// TIA Portal V20 export
FUNCTION_BLOCK "FB_PowerMeterSeq"   // FB92, SCL
{ S7_Optimized_Access := 'TRUE' }
// stored: AutoNumber false, MemoryReserve 100, SetENOAutomatically false
   VAR_INPUT
      iStartSeqCond : Bool;   // Start Sequence Conditions
      iJobReq : Bool;   // Job Request - From Main
      iPowerMeterHomePos : Bool;
      iPowerMeterWorkPos : Bool;
      iNC_Stopped : Bool;
      iPLC_DateAndTime : DTL;
      iStepPause : Bool;
      rMinValue : Real;
      rMaxValue : Real;
      iStopOption : Bool;
      rMeasureValue : Real;
      iMeasureDone : Bool;
   END_VAR
   VAR_OUTPUT
      oPowerMetertoHomeReq { ExternalAccessible := 'False'; ExternalVisible := 'False'; ExternalWritable := 'False'} : Bool;   // Shuttle Start Order - To FB_LoaderAxis
      oPowerMetertoWorkReq { ExternalAccessible := 'False'; ExternalVisible := 'False'; ExternalWritable := 'False'} : Bool;   // Shuttle Position Setpoint - To FB_LoaderAxis
      oStopNC_Req : Bool;
      oMsgBadMeasure : Bool;
      oStartMeasure : Bool;
      oStartArchive : Bool;
      oRID : Bool;
   END_VAR
   VAR
      sCurrent_Step_NB : Int;   // Active Step Number
      sCheck_Step_Condition : Bool;
      sOneStepForward : Bool;
      sRTOneStepForward : R_TRIG;
      sOneStepMode { S7_SetPoint := 'True'} : Bool;
      sStepForward : Bool;
      sInterface : "UDT_SequenceInterface";
      sPowerMetertoHomeReq { ExternalAccessible := 'False'; ExternalVisible := 'False'; ExternalWritable := 'False'} : Bool;
      sPowerMetertoWorkReq { ExternalAccessible := 'False'; ExternalVisible := 'False'; ExternalWritable := 'False'} : Bool;
      sStopNC_Req : Bool;
      sMsgBadMeasure : Bool;
      sStartMeasure : Bool;
      sStartArchive : Bool;
      sMeasureOK : Bool;
      sMeasureNOK : Bool;
      sRID : Bool;
      sHistory : Struct
         Activation : Bool;
         Steps : Array[0..99] of Int;
         Date_Time : Array[0..99] of DTL;
      END_STRUCT;
      StepText : "FB_GetTextErrorCode";
   END_VAR
   VAR_TEMP
      tIndex : Int;   // Index
   END_VAR
   VAR CONSTANT
      S00_INIT : Int := 0;
      S10_SET_RID : Int := 10;
      S20_POWERMETER_TO_WORK_POS : Int := 20;
      S30_START_MEASURE : Int := 30;
      S40_POWERMETER_TO_HOME_POS : Int := 40;
      S50_CHECK_MEASURE : Int := 50;
      S60_RESET_RID : Int := 60;
      S70_SPARE : Int := 70;
      S80_ARCHIVE_MEASURE : Int := 80;
      S160_RESET_RID : Int := 160;
      S170_STOP_CYCLE : Int := 170;
      S180_ARCHIVE_MEASURE : Int := 180;
      S295_JOB_DONE : Int := 295;
   END_VAR
   // StepText.sCode_error[0].ErrorCode := 0;
   // StepText.sCode_error[1].ErrorCode := 10;
   // StepText.sCode_error[2].ErrorCode := 20;
   // StepText.sCode_error[3].ErrorCode := 30;
   // StepText.sCode_error[4].ErrorCode := 40;
   // StepText.sCode_error[5].ErrorCode := 50;
   // StepText.sCode_error[6].ErrorCode := 60;
   // StepText.sCode_error[7].ErrorCode := 70;
   // StepText.sCode_error[8].ErrorCode := 80;
   // StepText.sCode_error[9].ErrorCode := 90;
   // StepText.sCode_error[10].ErrorCode := 95;
BEGIN
   REGION Description header 
       //==================================================================================
       // POSALUX Swiss SA / (C) Copyright 2026
       //----------------------------------------------------------------------------------
       // Title: FB_PowerMeterSeq
       // Comment/Function: 
       // Author: Fabien WALDT
       // Engineering: TIA Portal v20
       //----------------------------------------------------------------------------------
       // Change log table:
       // Version  | Date     | Expert in charge | Changes applied
       // ---------|----------|------------------|-----------------------------------------
       // 00.00.01 | 20260513 | WFA              | First released version
       // =================================================================================
   END_REGION

   REGION Define condition to start
       IF #iStartSeqCond THEN
           #sInterface.SequenceReleased := TRUE;
       ELSE
           // Standard sequencer controls
           #sInterface.SequenceReleased := FALSE;
           #sCurrent_Step_NB := #S00_INIT;
           #sInterface.SequenceRun := FALSE;
           #sInterface.JobDone := FALSE;
           #sCheck_Step_Condition := FALSE;

           // Dedicated sequencer controls
           #sPowerMetertoHomeReq := FALSE;
           #sPowerMetertoWorkReq := FALSE;
           #sStopNC_Req := FALSE;
           #sStartMeasure := FALSE;
           #sStartArchive := FALSE;
           #sMeasureOK := FALSE;
           #sMeasureNOK := FALSE;
           #sRID := FALSE;

           // Add specifics controls 
       END_IF;

       // Reset interface error
       IF #sInterface.Reset THEN
           #sInterface.Error := FALSE;
       END_IF;

       // One step forward
       #sRTOneStepForward.CLK := #sOneStepForward;
       #sRTOneStepForward();
       #sStepForward := (NOT #sOneStepMode OR (#sOneStepMode AND #sRTOneStepForward.Q)) AND NOT #iStepPause;
       #sOneStepForward := FALSE;

       // Action only true in dedicated steps
       #sStopNC_Req := FALSE;
       #sStartMeasure := FALSE;
   END_REGION

   REGION Sequence Function
       CASE #sCurrent_Step_NB OF
           #S00_INIT:
               REGION S00 INIT
                   #sCheck_Step_Condition := TRUE;
                   #sMsgBadMeasure := FALSE;
               END_REGION
           #S10_SET_RID:
               REGION S10_SET_RID
                   #sRID := TRUE;
                   #sCheck_Step_Condition := TRUE;
               END_REGION
           #S20_POWERMETER_TO_WORK_POS:
               REGION S20_POWERMETER_TO_WORK_POS
                   #sPowerMetertoHomeReq := FALSE;
                   #sPowerMetertoWorkReq := TRUE;
                   #sCheck_Step_Condition := TRUE;
               END_REGION
           #S30_START_MEASURE:
               REGION S30_START_MEASURE
                   #sStartMeasure := TRUE;
                   #sCheck_Step_Condition := TRUE;
               END_REGION
           #S40_POWERMETER_TO_HOME_POS:
               REGION S40_POWERMETER_TO_HOME_POS
                   #sPowerMetertoHomeReq := TRUE;
                   #sPowerMetertoWorkReq := FALSE;
                   #sCheck_Step_Condition := TRUE;
               END_REGION
           #S50_CHECK_MEASURE:
               REGION S50_WAIT_OPERATOR_RESTART
                   IF #rMeasureValue <= #rMaxValue AND #rMeasureValue >= #rMinValue THEN
                       #sMeasureOK := TRUE;
                       #sMeasureNOK := FALSE;
                   ELSE
                       #sMeasureOK := FALSE;
                       #sMeasureNOK := TRUE;
                   END_IF;
                   #sCheck_Step_Condition := TRUE;
               END_REGION
           #S60_RESET_RID:
               REGION S60_RESET_RID
                   #sRID := FALSE;
                   #sCheck_Step_Condition := TRUE;
               END_REGION
           #S70_SPARE:
               REGION S70_SPARE
                   #sCheck_Step_Condition := TRUE;
               END_REGION
           #S80_ARCHIVE_MEASURE:
               REGION S80_ARCHIVE_MEASURE
                   #sStartArchive := TRUE;
                   #sCheck_Step_Condition := TRUE;
               END_REGION

           #S160_RESET_RID:
               REGION S160_RESET_RID
                   #sRID := FALSE;
                   #sCheck_Step_Condition := TRUE;
               END_REGION
           #S170_STOP_CYCLE:
               REGION S170_STOP_CYCLE
                   #sStopNC_Req := TRUE;
                   #sCheck_Step_Condition := TRUE;
               END_REGION
           #S180_ARCHIVE_MEASURE:
               REGION S180_ARCHIVE_MEASURE
                   #sStartArchive := TRUE;
                   #sCheck_Step_Condition := TRUE;
               END_REGION

           #S295_JOB_DONE:
               REGION S295_JOB_DONE
                   #sInterface.JobDone := TRUE;
                   #sCheck_Step_Condition := TRUE;
               END_REGION
           ELSE:
               #sInterface.Error := TRUE;
       END_CASE;
   END_REGION

   REGION Sequence Next Step Condition
       IF #sCheck_Step_Condition THEN
           CASE #sCurrent_Step_NB OF
               #S00_INIT:
                   REGION S00 INIT
                       IF #sInterface.SequenceReleased AND #iJobReq THEN
                           #sCurrent_Step_NB := #S10_SET_RID;
                           #sInterface.SequenceRun := TRUE;
                           #sCheck_Step_Condition := FALSE;
                       ELSE
                           #sInterface.SequenceRun := FALSE;
                       END_IF;
                   END_REGION
               #S10_SET_RID:
                   REGION S10_SET_RID
                       IF #sInterface.SequenceReleased AND #sStepForward THEN
                           #sCurrent_Step_NB := #S20_POWERMETER_TO_WORK_POS;
                           #sCheck_Step_Condition := FALSE;
                       END_IF;
                   END_REGION
               #S20_POWERMETER_TO_WORK_POS:
                   REGION S20_POWERMETER_TO_WORK_POS
                       IF #sInterface.SequenceReleased AND #sStepForward AND #iPowerMeterWorkPos THEN
                           #sCurrent_Step_NB := #S30_START_MEASURE;
                           #sCheck_Step_Condition := FALSE;
                       END_IF;
                   END_REGION
               #S30_START_MEASURE:
                   REGION S30_START_MEASURE
                       IF #sInterface.SequenceReleased AND #sStepForward AND #iMeasureDone THEN
                           #sCurrent_Step_NB := #S40_POWERMETER_TO_HOME_POS;
                           #sCheck_Step_Condition := FALSE;
                       END_IF;
                   END_REGION
               #S40_POWERMETER_TO_HOME_POS:
                   REGION S40_POWERMETER_TO_HOME_POS
                       IF #sInterface.SequenceReleased AND #sStepForward AND #iPowerMeterHomePos THEN
                           #sCurrent_Step_NB := #S50_CHECK_MEASURE;
                           #sCheck_Step_Condition := FALSE;
                       END_IF;
                   END_REGION
                   #S50_CHECK_MEASURE:
                       REGION S50_CHECK_MEASURE
                           IF #sInterface.SequenceReleased AND #sStepForward AND (#sMeasureOK OR (#sMeasureNOK AND NOT #iStopOption)) THEN
                               #sCurrent_Step_NB := #S60_RESET_RID;
                               #sCheck_Step_Condition := FALSE;
                           ELSIF #sInterface.SequenceReleased AND #sStepForward AND (#sMeasureNOK AND #iStopOption) THEN
                               #sCurrent_Step_NB := #S160_RESET_RID;
                               #sCheck_Step_Condition := FALSE;
                           END_IF;
                       END_REGION
                   #S60_RESET_RID:
                       REGION S60_RESET_RID
                           IF #sInterface.SequenceReleased AND #sStepForward AND NOT #sRID THEN
                               #sCurrent_Step_NB := #S70_SPARE;
                               #sCheck_Step_Condition := FALSE;
                           END_IF;
                       END_REGION
                   #S70_SPARE:
                       REGION S70_SPARE
                           IF #sInterface.SequenceReleased AND #sStepForward AND "AlwaysTRUE" THEN
                               #sCurrent_Step_NB := #S80_ARCHIVE_MEASURE;
                               #sCheck_Step_Condition := FALSE;
                           END_IF;
                       END_REGION
                   #S80_ARCHIVE_MEASURE:
                       REGION S80_ARCHIVE_MEASURE
                           IF #sInterface.SequenceReleased AND #sStepForward AND "AlwaysTRUE" THEN
                               #sCurrent_Step_NB := #S295_JOB_DONE;
                               #sCheck_Step_Condition := FALSE;
                           END_IF;
                       END_REGION

                   #S160_RESET_RID:
                       REGION S160_RESET_RID
                           IF #sInterface.SequenceReleased AND #sStepForward AND NOT #sRID THEN
                               #sCurrent_Step_NB := #S170_STOP_CYCLE;
                               #sCheck_Step_Condition := FALSE;
                           END_IF;
                       END_REGION
                   #S170_STOP_CYCLE:
                       REGION S170_STOP_CYCLE
                           IF #sInterface.SequenceReleased AND #sStepForward AND #iNC_Stopped THEN
                               #sCurrent_Step_NB := #S180_ARCHIVE_MEASURE;
                               #sCheck_Step_Condition := FALSE;
                           END_IF;
                       END_REGION
                   #S180_ARCHIVE_MEASURE:
                       REGION S180_ARCHIVE_MEASURE
                           IF #sInterface.SequenceReleased AND #sStepForward AND "AlwaysTRUE" THEN
                               #sCurrent_Step_NB := #S295_JOB_DONE;
                               #sCheck_Step_Condition := FALSE;
                           END_IF;
                       END_REGION

                       #S295_JOB_DONE:
                           REGION S295_JOB_DONE
                               IF NOT #iJobReq THEN
                                   #sCurrent_Step_NB := #S00_INIT;
                                   #sCheck_Step_Condition := FALSE;
                                   #sInterface.JobDone := FALSE;
                               END_IF;
                           END_REGION
               ELSE
                   #sInterface.Error := TRUE;
           END_CASE;
       END_IF;
   END_REGION

   REGION Outputs Update
       #oPowerMetertoHomeReq := #sPowerMetertoHomeReq;
       #oPowerMetertoWorkReq := #sPowerMetertoWorkReq;
       #oStopNC_Req := #sStopNC_Req;
       #oMsgBadMeasure := #sMsgBadMeasure;
       #oStartMeasure := #sStartMeasure;
       #oStartArchive := #sStartArchive;
       #oRID := #sRID;
   END_REGION

   REGION Steps - Date and Time History
       IF #sHistory.Activation THEN
           IF #sHistory.Steps[0] <> #sCurrent_Step_NB THEN
               FOR #tIndex := 98 TO 0 BY -1 DO
                   #sHistory.Steps[#tIndex + 1] := #sHistory.Steps[#tIndex];
                   #sHistory.Date_Time[#tIndex + 1] := #sHistory.Date_Time[#tIndex];
               END_FOR;
               #sHistory.Steps[0] := #sCurrent_Step_NB;
               #sHistory.Date_Time[0] := #iPLC_DateAndTime;
           END_IF;
       END_IF;
   END_REGION

   REGION Steps Text
       #StepText(iErrorCode := #sCurrent_Step_NB,
                 oErrorText => #StepText.oErrorText);
   END_REGION
END_FUNCTION_BLOCK
